INTERFACE PUBLIC I_MoveCommand EXTENDS I_AsyncCommand

PROPERTY PUBLIC IsActive : BOOL
GET // PUBLIC
END_GET
END_PROPERTY

END_INTERFACE

(* stored: Version 1.1.0.1, ProductVersion 3.1.4024.12
   Itf I_MoveCommand: Id {ace235f2-e3c9-4384-9979-8089e1813370}
   Property IsActive: Id {7440f60b-eea9-007f-0eeb-decc794bf55c}
   Get Get: Id {0357b9df-10e9-063d-046c-748ce5aac12b} *)
